/// Provides error codes for TcLogCore
{attribute 'qualified_only'}
{attribute 'strict'}
{attribute 'to_string'}
TYPE ErrorCodes : 
(
	None := 0,
	OpeningFileFailed,
	WritingToFileFailed,
	ClosingFileFailed,
	EnumeratingFilesInSpecifiedDirectoryFailed,
	DeletingFileFailed,
	FifoOverflow
);
END_TYPE

(* stored: Version 1.1.0.1, ProductVersion 3.1.4024.12
   DUT ErrorCodes: Id {0e8d414f-7d83-44fd-bab7-2f3442435cad} *)
